ABB RAPID module: Wizard.modx

MODULE Wizard
PERS robtarget Location1:=[[-336.349548339844, 0.510710597038269, 992.6142578125], [0.363380044698715, 0.264791667461395, -0.886605024337769, -0.108498312532902], [1, 2, -1, 1], [9000000000, 9000000000, 9000000000, 9000000000, 9000000000, 9000000000]];
PERS robtarget Location2:=[[-798.059631347656, 20.9319171905518, 767.132263183594], [0.65837174654007, 0.198111280798912, -0.696351647377014, -0.205895528197289], [1, 2, -1, 1], [9000000000, 9000000000, 9000000000, 9000000000, 9000000000, 9000000000]];
PERS robtarget Location3:=[[-518.156921386719, 154.585983276367, 970.468688964844], [0.591564536094666, 0.110178925096989, -0.749538600444794, -0.275869369506836], [1, 1, -1, 1], [9000000000, 9000000000, 9000000000, 9000000000, 9000000000, 9000000000]];
PERS robtarget Location4:=[[-627.505249023438, 193.126693725586, 711.158386230469], [0.075685434043407, 0.140533089637756, -0.986474812030792, -0.0372767299413681], [1, 1, -1, 1], [9000000000, 9000000000, 9000000000, 9000000000, 9000000000, 9000000000]];
PERS robtarget O1:=[[356.637451171875, 161.037048339844, 513.128356933594], [0.0388496816158295, -0.776131391525269, -0.358248889446259, -0.517463564872742], [0, 1, 0, 1], [9000000000, 9000000000, 9000000000, 9000000000, 9000000000, 9000000000]];
PERS robtarget O2:=[[356.619445800781, 121.282089233398, 484.093872070313], [0.00313940364867449, -0.806082367897034, -0.327470064163208, -0.492934823036194], [0, 1, 0, 1], [9000000000, 9000000000, 9000000000, 9000000000, 9000000000, 9000000000]];
PERS robtarget O3:=[[399.640594482422, 143.169784545898, 468.373107910156], [0.00769960461184382, 0.794183015823364, 0.382436096668243, 0.472182840108871], [0, 1, 0, 1], [9000000000, 9000000000, 9000000000, 9000000000, 9000000000, 9000000000]];
PERS robtarget O4:=[[436.398681640625, 185.750854492188, 440.245086669922], [0.083333015441895, -0.836603939533234, -0.298512071371078, -0.451707899570465], [0, 1, 0, 1], [9000000000, 9000000000, 9000000000, 9000000000, 9000000000, 9000000000]];
PERS robtarget O5:=[[384.975860595703, 184.290008544922, 436.962097167969], [0.130016103386879, -0.904695689678192, -0.099378101527691, -0.393377006053925], [0, 1, 0, 1], [9000000000, 9000000000, 9000000000, 9000000000, 9000000000, 9000000000]];
PERS robtarget P1:=[[555.272094726563, 252.178009033203, 617.894104003906], [0.081425286829472, 0.61410117149353, -0.783669710159302, -0.0459511838853359], [0, 0, -1, 0], [9000000000, 9000000000, 9000000000, 9000000000, 9000000000, 9000000000]];
PERS robtarget P2:=[[581.155456542969, 294.388061523438, 592.781372070313], [0.188104867935181, 0.633526146411896, -0.750378608703613, 0.0138965677469969], [0, -1, -1, 0], [9000000000, 9000000000, 9000000000, 9000000000, 9000000000, 9000000000]];
PERS robtarget P3:=[[600.000305175781, 305.776336669922, 591.8310546875], [0.121595151722431, 0.64362096786499, -0.755053102970123, 0.0293502137064934], [0, -1, -1, 0], [9000000000, 9000000000, 9000000000, 9000000000, 9000000000, 9000000000]];
PERS robtarget P4:=[[553.178527832031, 356.432434082031, 589.507019042969], [0.16638009250164, 0.676077246665955, -0.716881811618805, 0.0363007448613644], [0, -1, -1, 0], [9000000000, 9000000000, 9000000000, 9000000000, 9000000000, 9000000000]];
PERS robtarget P5:=[[432.768585205078, 238.302230834961, 615.04248046875], [0.0402561873197556, -0.661645650863647, 0.747375845909119, -0.0450976602733135], [0, -1, -1, 0], [9000000000, 9000000000, 9000000000, 9000000000, 9000000000, 9000000000]];
PERS robtarget P6:=[[475.761413574219, 225.393676757813, 604.477722167969], [0.0422640293836594, -0.645888447761536, 0.75911670923233, -0.06916418671608], [0, -1, -1, 0], [9000000000, 9000000000, 9000000000, 9000000000, 9000000000, 9000000000]];
PERS robtarget P7:=[[469.6630859375, 219.079544067383, 598.929931640625], [0.066877692937851, -0.600106239318848, 0.795571863651276, 0.049651961773634], [0, 0, -1, 0], [9000000000, 9000000000, 9000000000, 9000000000, 9000000000, 9000000000]];
PERS robtarget Q1:=[[528.979309082031, 222.100708007813, 673.107788085938], [0.0288146324455738, 0.59828782081604, -0.797598898410797, -0.071115754544735], [0, 0, -1, 0], [9000000000, 9000000000, 9000000000, 9000000000, 9000000000, 9000000000]];
PERS robtarget Q2:=[[527.635681152344, 221.418273925781, 659.507080078125], [0.0496013537049294, 0.603277981281281, -0.794661700725555, -0.045915212482214], [0, 0, -1, 0], [9000000000, 9000000000, 9000000000, 9000000000, 9000000000, 9000000000]];
PERS robtarget Q3:=[[534.149780273438, 236.523788452148, 635.858581542969], [0.0582736246287823, 0.623373210430145, -0.779543697834015, 0.0179351884871721], [0, -1, -1, 0], [9000000000, 9000000000, 9000000000, 9000000000, 9000000000, 9000000000]];
PERS robtarget Q4:=[[547.385986328125, 245.032989501953, 635.38818359375], [0.0130515284836292, 0.624627470970154, -0.780573189258575, 0.0193815547972918], [0, -1, -1, 0], [9000000000, 9000000000, 9000000000, 9000000000, 9000000000, 9000000000]];
PERS robtarget Q5:=[[532.101745605469, 251.928833007813, 629.298828125], [0.0255458690226078, 0.616161584854126, -0.785374164581299, -0.0536635741591454], [0, 0, -1, 0], [9000000000, 9000000000, 9000000000, 9000000000, 9000000000, 9000000000]];
	PROC main()
  <SMT>
	ENDPROC
ENDMODULE
